{attribute addProperty BoxType "EL6201-0000-0017"}
{attribute addProperty Id "Slave_19A_DO0BIT10.125145Slave_19A_DO1BIT10.125146Slave_19A_DO2BIT10.125147Slave_19A_DO3BIT10.125148Slave_19B_DO0BIT10.125149Slave_19B_DO1BIT10.125150Slave_19B_DO2BIT10.125151Slave_19B_DO3BIT10.125152"}
{attribute addProperty CRC "1517220697"}
{attribute addProperty SizeInBites "8"}
{attribute addProperty SizeInBytes "1"}
TYPE Slave_19_Outputs_5A6EF359 :
STRUCT
	{attribute addProperty Name "Slave_19A_DO0"}
	Slave_19A_DO0 : BIT;
	{attribute addProperty Name "Slave_19A_DO1"}
	Slave_19A_DO1 : BIT;
	{attribute addProperty Name "Slave_19A_DO2"}
	Slave_19A_DO2 : BIT;
	{attribute addProperty Name "Slave_19A_DO3"}
	Slave_19A_DO3 : BIT;
	{attribute addProperty Name "Slave_19B_DO0"}
	Slave_19B_DO0 : BIT;
	{attribute addProperty Name "Slave_19B_DO1"}
	Slave_19B_DO1 : BIT;
	{attribute addProperty Name "Slave_19B_DO2"}
	Slave_19B_DO2 : BIT;
	{attribute addProperty Name "Slave_19B_DO3"}
	Slave_19B_DO3 : BIT;
END_STRUCT
END_TYPE

(* stored: Version 1.2.0.0, ProductVersion 3.1.4024.9
   DUT Slave_19_Outputs_5A6EF359: Id {c4288155-4013-46c5-aa9b-f4c0eb61c9b6} *)
